FUNCTION_BLOCK Auto_ColorDetection
VAR_INPUT
	ColorSensor: INT;
	ColorCode_1: INT;
	ColorCode_2: INT;
	ColorCode_3: INT;
END_VAR
VAR_OUTPUT
	Color_1: BOOL;
	Color_2: BOOL;
	Color_3: BOOL;
END_VAR
VAR

END_VAR

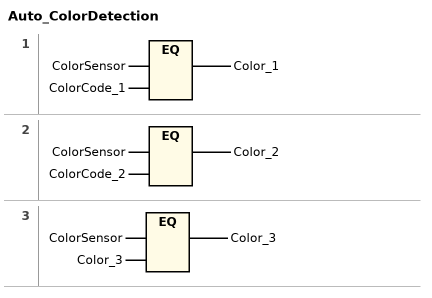
// NETWORK 1
Color_1 := ColorSensor = ColorCode_1;

// NETWORK 2
Color_2 := ColorSensor = ColorCode_2;

// NETWORK 3
Color_3 := ColorSensor = Color_3;

END_FUNCTION_BLOCK

(* stored: Version 1.1.0.1, ProductVersion 3.1.4024.15
   POU Auto_ColorDetection: Id {f042d649-19e0-4dea-a103-0ed2ef0d7010}, SpecialFunc None *)
